// TIA Portal V17 export
// export: Created 2022-07-20T07:02:37.8832777Z, ExportSetting WithDefaults, DisplayName Totally Integrated Automation Portal, DisplayVersion V17, DisplayName TIA Portal Openness, DisplayVersion V17, DisplayName TIA Portal Version Control Interface, DisplayVersion V17, DisplayName SINAMICS Startdrive Advanced, DisplayVersion V17, DisplayName SINAMICS Startdrive G130, G150, S120, S150, SINAMICS MV, S210, DisplayVersion V17, DisplayName SINAMICS Startdrive G110M, G120, G120C, G120D, G120P, G115D, DisplayVersion V17, DisplayName STEP 7 Professional, DisplayVersion V17, DisplayName STEP 7 Safety, DisplayVersion V17, DisplayName WinCC Advanced, DisplayVersion V17
VAR_GLOBAL   // PLC tag table "SolenoidValve_SMC_CommunicationTable"
   SMC_1_Input_1 AT %IB38 : Byte;
   SMC_1_Input_2 AT %IB39 : Byte;
   SMC_1_Input_3 AT %IB40 : Byte;
   SMC_1_Input_4 AT %IB41 : Byte;
   SMC_1_Output_1 AT %QB490 : Byte;
   SMC_1_Output_2 AT %QB491 : Byte;
   SMC_1_Output_3 AT %QB492 : Byte;
   SMC_1_Output_4 AT %QB493 : Byte;
END_VAR
